{attribute 'linkalways'} 
{attribute 'no_explicit_call' := 'This FB is a CLASS and must be accessed using methods or properties'}
{attribute 'enable_dynamic_creation'}
FUNCTION_BLOCK FINAL ADD_USINT EXTENDS Node
VAR
	in1 : _USINT(0);
	in2 : _USINT(0);
	out : _USINT(0);
END_VAR

METHOD PUBLIC Clone : I_Node
VAR
	pNode : POINTER TO ADD_USINT;
END_VAR
pNode := __NEW(ADD_USINT);
Clone := pNode^;
END_METHOD

METHOD FB_init : BOOL
VAR_INPUT
	bInitRetains : BOOL; // if TRUE, the retain variables are initialized (warm start / cold start)
	bInCopyCode : BOOL;  // if TRUE, the instance afterwards gets moved into the copy code (online change)
END_VAR
AddInput('in1',THIS^.in1);
AddInput('in2',THIS^.in2);
AddOutput('out', THIS^.out);
END_METHOD

METHOD PROTECTED OnExecute
VAR
END_VAR
out.Value := in1.Value + in2.Value;
END_METHOD

END_FUNCTION_BLOCK

(* stored: Version 1.1.0.1, ProductVersion 3.1.4024.15
   POU ADD_USINT: Id {e8a6293b-452c-43a1-9960-6767466289ed}, SpecialFunc None
   Folder Constructor: Id {e0ba873a-efed-4217-a1c5-93051b21021c}
   Method Clone: Id {9f80997f-f2d8-4d6b-ac42-7bbf9fb593a1}
   Method FB_init: Id {db4481e9-05f9-4d31-bb2f-680042a3697f}
   Method OnExecute: Id {c323de3a-4e4e-4ab5-8ae5-4677584c5b39} *)
